Staubli VAL3: PE_Solar.pjx

--- PE_Solar.pjx ---
Parameters version=s7.8.3 stackSize=10000 millimeterUnit=true
Program file=init.pgx
Program file=libload.pgx
Program file=start.pgx
Program file=stop.pgx
Program file=WatchDog.pgx
Data file=PE_Solar.dtx
Library alias=page_view path=Disk://page/page_viewTraj/page_viewTraj.pjx
Library alias=pub path=Disk://public_temp/pub/pub.pjx
Library alias=cycle path=Disk://cycle/cycle.pjx
Library alias=io path=Disk://io/io.pjx

--- start.pgx ---
program start()
begin

  call init()
  taskCreate "PLC",100,cycle:_tPLC()
  taskCreate "HIM",100,libload("Disk://page/page_viewTraj")
  taskCreate "_WatchDog",100,cycle:_WatchDog()
  // call WatchDog()

end

--- init.pgx ---
program init()
begin
  io:sToShow="程序复位，准备开始"
end

--- libload.pgx ---
program libload(string s_Item (dimensions=1))
begin
  pub:libLoad(s_Item)
  call pub:main()
end

--- WatchDog.pgx ---
program WatchDog()
begin
end
